// TIA Portal V20 export
DATA_BLOCK "DB_FeedOverride"   // DB116
// stored: InstanceOfName FB_FeedOverride, InstanceOfType FB
"FB_FeedOverride"
   // VAR_INPUT
   //    iA_FD_OR : Byte;
   // END_VAR
   // VAR_OUTPUT
   //    oFeedOverride : Byte;
   // END_VAR
BEGIN
END_DATA_BLOCK
